// SIMATIC S7-200 SMART project (STEP 7-Micro/WIN SMART), CPU ST40

SYMBOL_TABLE System Symbols
Always_On        SM0.0    // Always ON
First_Scan_On    SM0.1    // ON for the first scan cycle only
Clock_1s         SM0.5    // Clock pulse that is ON for 0.5 s, OFF for 0.5 s, for a duty cycle time of 1 s.
END_SYMBOL_TABLE

ORGANIZATION_BLOCK MAIN:OB1
TITLE=Program Comments
BEGIN
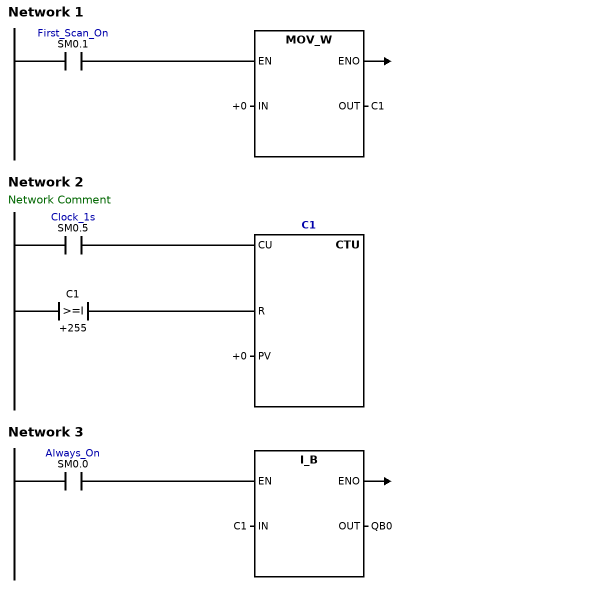
Network 1
LD     First_Scan_On:SM0.1
MOVW   +0, C1
Network 2
// Network Comment
LD     Clock_1s:SM0.5
LDW>=  C1, +255
CTU    C1, +0
Network 3
LD     Always_On:SM0.0
ITB    C1, QB0
END_ORGANIZATION_BLOCK
